// TIA Portal V18 export
FUNCTION "FC_LadDemo" : Void   // FC1, LAD
{ S7_Optimized_Access := 'TRUE' }
   VAR_INPUT
      In1 : Bool;
   END_VAR
BEGIN

REGION Network 1
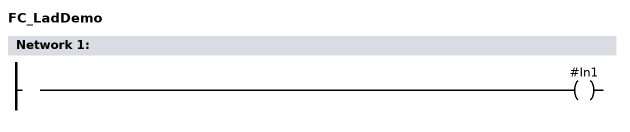
   #In1 := TRUE;
END_REGION
END_FUNCTION
